(* CoDeSys 2.3 library: mod_com.lib *)

(* Data type *)
(* Additional information  *)
TYPE ADD_DESC :

STRUCT
	posPAA : WORD;    (* Position of this module in the output process image (PLC) [bits] *)
	posPAE : WORD;    (* Position of this module in the input process image (PLC) [bits] *)
	sizePAA : BYTE;       (* Number of bits in the output process image (PLC) *)
	sizePAE : BYTE;       (* Number of bits in the input process image (PLC) *)
	channels : BYTE;     (* Number of channels (only for complex modules) *)
	altFormat : BYTE;    (* Alternative format *)
END_STRUCT

END_TYPE

(* Data type *)
(* Information of a module *)
TYPE MODULE_INFO :

STRUCT
	physicalPos : BYTE;     (* Physical position of the module *)
	moduleType : WORD;  (* Number of the module 750-xxx *)
	desc : ADD_DESC;      (* Additional information *)
END_STRUCT

END_TYPE


(*   remark
	-------------------------------------------

	'moduleType' for digital modules:

	16#00D0:  no data in the input and output process image (PLC)
	16#00D1:  data only in the input process image (PLC)
	16#00D2:  data only in the output process image (PLC)
	16#00D3:  data in the input and output process image (PLC)

*)

(* Data type *)
(* Type of the access *)
TYPE MODULE_INFO_ACCESS :

STRUCT
	physicalPosOf : BYTE;     (* Start of the physical position *)
	physicalPosTo : BYTE;    (* End of the physical position *)
	typeNumber : BYTE;         (* Wich number of the module type is meant *)
	moduleType : WORD;      (* module type *)
	window : WORD;               (* Window for 'moduleType' in ascending direction *)
END_STRUCT

END_TYPE


(*    Access methods:
	------------------------------------------------------------------------------------------------------
	physicalPosTo <> 0:

		Information of the modules from 'physicalPosOf' to 'physicalPosTo'
	------------------------------------------------------------------------------------------------------
	physicalPosTo = 0 AND moduleType <> 0 (only for complex modules):

		Information of the module (typeNumber) of the type 'moduleType' + ' window'
	------------------------------------------------------------------------------------------------------
	physicalPosTo = 0 AND moduleType = 0:

		Information of all modules
*)

(* POU SET_DIGITAL_INPUT_OFFSET, IL *)
FUNCTIONBLOCK  SET_DIGITAL_INPUT_OFFSET
(* set digital input bits offset *)
VAR_INPUT
	EN: BOOL;
	DIG_IN_OFFSET:WORD;
END_VAR
VAR_OUTPUT
	ENO: BOOL;
	ERROR:WORD;
END_VAR
	LD		0
END_FUNCTION_BLOCK

(* POU SET_DIGITAL_OUTPUT_OFFSET, IL *)
FUNCTIONBLOCK SET_DIGITAL_OUTPUT_OFFSET
(* set digital output bits offset *)
VAR_INPUT
	EN: BOOL;
	DIG_OUT_OFFSET:WORD;
END_VAR
VAR_OUTPUT
	ENO: BOOL;
	ERROR:WORD;
END_VAR
	LD		0
END_FUNCTION_BLOCK

(* POU ADD_PI_INFORMATION, IL *)
(* Additional Process Image Information of modules *)
FUNCTION ADD_PI_INFORMATION : BOOL

VAR_INPUT
	EN : BOOL;
	pAccess : POINTER TO MODULE_INFO_ACCESS;
	pInfo : POINTER TO MODULE_INFO;
END_VAR

VAR
END_VAR


(*   Example
	-------------------------------------------------------------------
	VAR
		access : MODULE_INFO_ACCESS;
		info : ARRAY[0..63] OF MODULE_INFO;
	END_VAR

	access.physicalPosTo := 0;
	access.moduleType := 0;

	ADD_PI_INFORMATION( 1, ADR(access), ADR(info[0]) );
*)
LD 1
END_FUNCTION

(* POU CRC16, IL *)
FUNCTION_BLOCK CRC16
VAR
	CRCHI: BYTE;
	CRCLO: BYTE;
	INDEX: BYTE;
	STATE: BYTE;
END_VAR
VAR_INPUT
	INPUT: BYTE;
	EN: BOOL;
END_VAR
VAR_OUTPUT
	CRC: WORD;
END_VAR
LD 0
END_FUNCTION_BLOCK

(* POU FBUS_ERROR_INFORMATION, IL *)
FUNCTION_BLOCK FBUS_ERROR_INFORMATION
VAR_OUTPUT
	FBUS_ERROR: BOOL;
	ERROR: WORD;
END_VAR
LD 0
END_FUNCTION_BLOCK

(* POU GET_DIGITAL_INPUT_OFFSET, IL *)
FUNCTION_BLOCK GET_DIGITAL_INPUT_OFFSET
VAR_OUTPUT
	DIG_IN_OFFSET: WORD;
	ERROR: WORD;
END_VAR
LD 0
END_FUNCTION_BLOCK

(* POU GET_DIGITAL_OUTPUT_OFFSET, IL *)
FUNCTION_BLOCK GET_DIGITAL_OUTPUT_OFFSET
VAR_OUTPUT
	DIG_OUT_OFFSET: WORD;
	ERROR: WORD;
END_VAR
LD 0
END_FUNCTION_BLOCK

(* POU KBUS_ERROR_INFORMATION, IL *)
FUNCTION_BLOCK KBUS_ERROR_INFORMATION
VAR_OUTPUT
	KBUS_ERROR: BOOL;
	BITLEN: WORD;
	TERMINALS: WORD;
	RESERVED1: WORD;
	RESERVED2: WORD;
	FAIL_ADDRESS: WORD;
END_VAR
LD 0
END_FUNCTION_BLOCK

(* POU MOD_COM_VERSION, IL *)
FUNCTION MOD_COM_VERSION : WORD
VAR_INPUT
	EN: BOOL;
END_VAR
LD 0
END_FUNCTION

(* POU PI_INFORMATION, IL *)
FUNCTION_BLOCK PI_INFORMATION
VAR_OUTPUT
	ANALOG_OUTLENGTH: WORD;
	ANALOG_INLENGTH: WORD;
	DIGITAL_OUTLENGTH: WORD;
	DIGITAL_INLENGTH: WORD;
	OUTPUTBITS_OFFSET: WORD;
	INPUTBITS_OFFSET: WORD;
END_VAR
LD 0
END_FUNCTION_BLOCK

(* POU READ_INPUT_BIT, IL *)
FUNCTION_BLOCK READ_INPUT_BIT
VAR_INPUT
	WORD_ADDRESS: WORD;
	BIT_ADDRESS: WORD;
END_VAR
VAR_OUTPUT
	VALUE: BOOL;
	ERROR: BOOL;
END_VAR
LD 0
END_FUNCTION_BLOCK

(* POU READ_INPUT_WORD, IL *)
FUNCTION_BLOCK READ_INPUT_WORD
VAR_INPUT
	WORD_ADDRESS: WORD;
END_VAR
VAR_OUTPUT
	VALUE: WORD;
	ERROR: BOOL;
END_VAR
LD 0
END_FUNCTION_BLOCK

(* POU READ_OUTPUT_BIT, IL *)
FUNCTION_BLOCK READ_OUTPUT_BIT
VAR_INPUT
	WORD_ADDRESS: WORD;
	BIT_ADDRESS: WORD;
END_VAR
VAR_OUTPUT
	VALUE: BOOL;
	ERROR: BOOL;
END_VAR
LD 0
END_FUNCTION_BLOCK

(* POU READ_OUTPUT_WORD, IL *)
FUNCTION_BLOCK READ_OUTPUT_WORD
VAR_INPUT
	WORD_ADDRESS: WORD;
END_VAR
VAR_OUTPUT
	VALUE: WORD;
	ERROR: BOOL;
END_VAR
LD 0
END_FUNCTION_BLOCK

(* POU SLAVE_ADDRESS, IL *)
FUNCTION_BLOCK SLAVE_ADDRESS
VAR_OUTPUT
	SLAVE_ADDRESS: BYTE;
END_VAR
LD 0
END_FUNCTION_BLOCK

(* POU WRITE_OUTPUT_BIT, IL *)
FUNCTION_BLOCK WRITE_OUTPUT_BIT
VAR_INPUT
	WORD_ADDRESS: WORD;
	BIT_ADDRESS: WORD;
	VALUE: BOOL;
END_VAR
VAR_OUTPUT
	ERROR: BOOL;
END_VAR
LD 0
END_FUNCTION_BLOCK

(* POU WRITE_OUTPUT_WORD, IL *)
FUNCTION_BLOCK WRITE_OUTPUT_WORD
VAR_INPUT
	WORD_ADDRESS: WORD;
	VALUE: WORD;
END_VAR
VAR_OUTPUT
	ERROR: BOOL;
END_VAR
LD 0
END_FUNCTION_BLOCK
